FUNCTION F_ValveClear : bool
VAR_INPUT
	Input																: BOOL;
	Open																: BOOL;
	Closed																: BOOL;
END_VAR
VAR
END_VAR

// F_ValveClear
// Rev 1.0 - December 28, 2023

F_ValveClear															:= ((Input AND Open) OR (NOT Input AND Closed)) AND NOT (Open = Closed);

END_FUNCTION

(* stored: Version 1.1.0.1, ProductVersion 3.1.4024.12
   POU F_ValveClear: Id {7a1dd4b2-7dbb-4250-9f37-31cd86071f1d}, SpecialFunc None *)
